% RSLogix 500 project I2P JOB 23 - SOLUTION_BAK116.RSS, saved by version 10.00.00.00 %
PROJECT "MLO2B"    % processor: Bul.1763 MicroLogix 1100 Series B %

PROGRAM FILES
  LAD 2   18 rungs

DATA FILES
  O0 OUTPUT  4 elements
  I1 INPUT  6 elements
  S2 STATUS  66 elements
  B3 BINARY  1 elements
  T4 TIMER  2 elements
  C5 COUNTER  2 elements
  R6 CONTROL  1 elements
  N7 INTEGER  2 elements
  F8 FLOAT  1 elements

LADDER 2
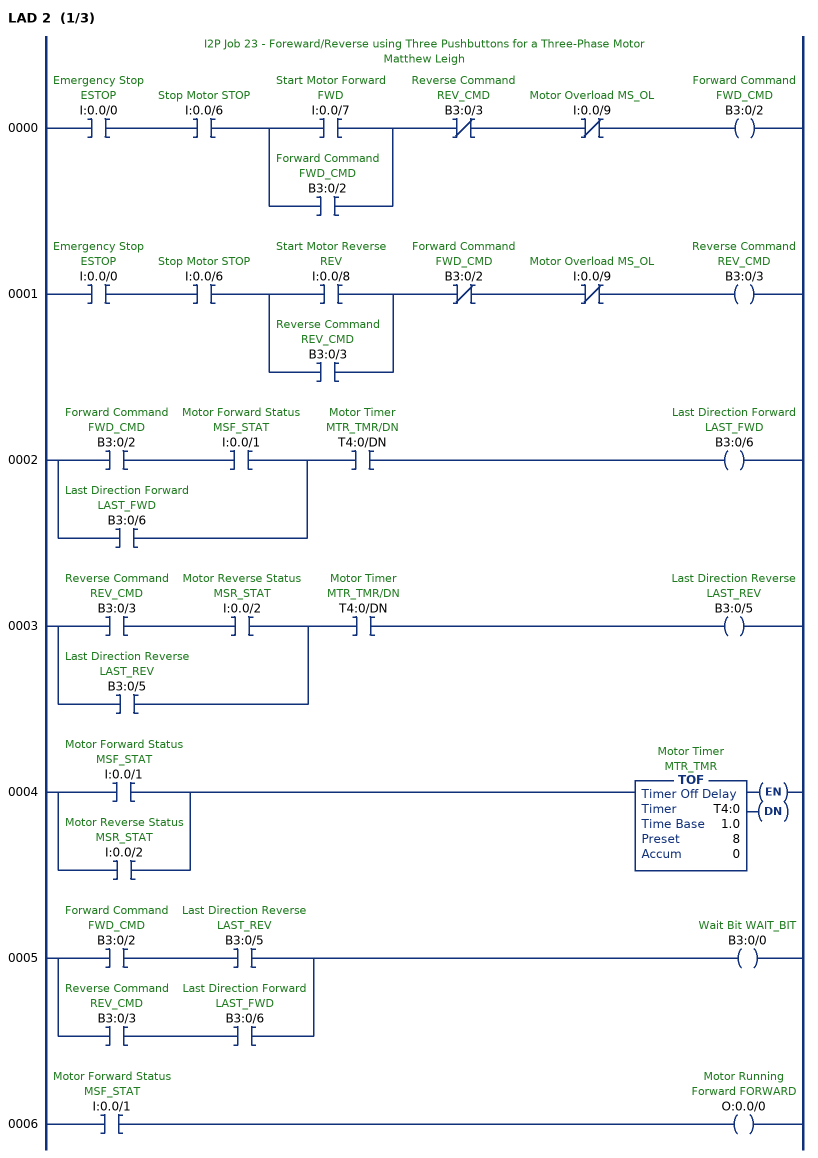
% Rung: 0 %
% I2P Job 23 - Foreward/Reverse using Three Pushbuttons for a Three-Phase Motor
% Matthew Leigh %
SOR XIC I:0.0/0 XIC I:0.0/6 BST XIC I:0.0/7 NXB XIC B3:0/2 BND XIO B3:0/3 XIO I:0.0/9 OTE B3:0/2 EOR
%   I:0.0/0  ESTOP  "Emergency Stop" %
%   I:0.0/6  STOP  "Stop Motor" %
%   I:0.0/7  FWD  "Start Motor Forward" %
%   B3:0/2  FWD_CMD  "Forward Command" %
%   B3:0/3  REV_CMD  "Reverse Command" %
%   I:0.0/9  MS_OL  "Motor Overload" %
% Rung: 1 %
SOR XIC I:0.0/0 XIC I:0.0/6 BST XIC I:0.0/8 NXB XIC B3:0/3 BND XIO B3:0/2 XIO I:0.0/9 OTE B3:0/3 EOR
%   I:0.0/0  ESTOP  "Emergency Stop" %
%   I:0.0/6  STOP  "Stop Motor" %
%   I:0.0/8  REV  "Start Motor Reverse" %
%   B3:0/3  REV_CMD  "Reverse Command" %
%   B3:0/2  FWD_CMD  "Forward Command" %
%   I:0.0/9  MS_OL  "Motor Overload" %
% Rung: 2 %
SOR BST XIC B3:0/2 XIC I:0.0/1 NXB XIC B3:0/6 BND XIC T4:0/DN OTE B3:0/6 EOR
%   B3:0/2  FWD_CMD  "Forward Command" %
%   I:0.0/1  MSF_STAT  "Motor Forward Status" %
%   B3:0/6  LAST_FWD  "Last Direction Forward" %
%   T4:0  MTR_TMR  "Motor Timer" %
% Rung: 3 %
SOR BST XIC B3:0/3 XIC I:0.0/2 NXB XIC B3:0/5 BND XIC T4:0/DN OTE B3:0/5 EOR
%   B3:0/3  REV_CMD  "Reverse Command" %
%   I:0.0/2  MSR_STAT  "Motor Reverse Status" %
%   B3:0/5  LAST_REV  "Last Direction Reverse" %
%   T4:0  MTR_TMR  "Motor Timer" %
% Rung: 4 %
SOR BST XIC I:0.0/1 NXB XIC I:0.0/2 BND TOF T4:0 1.0 8 0 EOR
%   I:0.0/1  MSF_STAT  "Motor Forward Status" %
%   I:0.0/2  MSR_STAT  "Motor Reverse Status" %
%   T4:0  MTR_TMR  "Motor Timer" %
% Rung: 5 %
SOR BST XIC B3:0/2 XIC B3:0/5 NXB XIC B3:0/3 XIC B3:0/6 BND OTE B3:0/0 EOR
%   B3:0/2  FWD_CMD  "Forward Command" %
%   B3:0/5  LAST_REV  "Last Direction Reverse" %
%   B3:0/3  REV_CMD  "Reverse Command" %
%   B3:0/6  LAST_FWD  "Last Direction Forward" %
%   B3:0/0  WAIT_BIT  "Wait Bit" %
% Rung: 6 %
SOR XIC I:0.0/1 OTE O:0.0/0 EOR
%   I:0.0/1  MSF_STAT  "Motor Forward Status" %
%   O:0.0/0  FORWARD  "Motor Running Forward" %

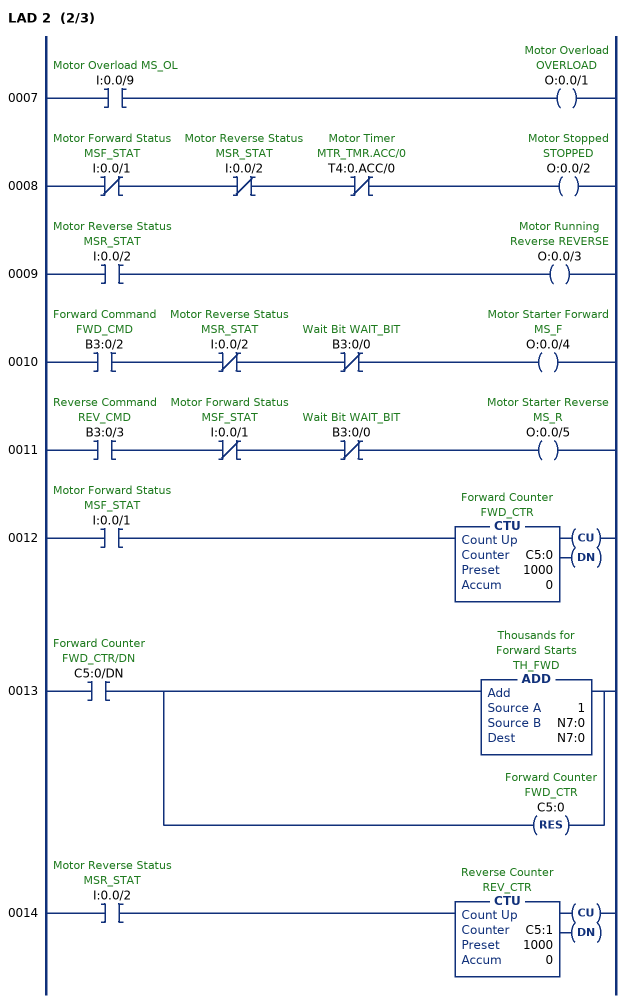
% Rung: 7 %
SOR XIC I:0.0/9 OTE O:0.0/1 EOR
%   I:0.0/9  MS_OL  "Motor Overload" %
%   O:0.0/1  OVERLOAD  "Motor Overload" %
% Rung: 8 %
SOR XIO I:0.0/1 XIO I:0.0/2 XIO T4:0.ACC/0 OTE O:0.0/2 EOR
%   I:0.0/1  MSF_STAT  "Motor Forward Status" %
%   I:0.0/2  MSR_STAT  "Motor Reverse Status" %
%   T4:0  MTR_TMR  "Motor Timer" %
%   O:0.0/2  STOPPED  "Motor Stopped" %
% Rung: 9 %
SOR XIC I:0.0/2 OTE O:0.0/3 EOR
%   I:0.0/2  MSR_STAT  "Motor Reverse Status" %
%   O:0.0/3  REVERSE  "Motor Running Reverse" %
% Rung: 10 %
SOR XIC B3:0/2 XIO I:0.0/2 XIO B3:0/0 OTE O:0.0/4 EOR
%   B3:0/2  FWD_CMD  "Forward Command" %
%   I:0.0/2  MSR_STAT  "Motor Reverse Status" %
%   B3:0/0  WAIT_BIT  "Wait Bit" %
%   O:0.0/4  MS_F  "Motor Starter Forward" %
% Rung: 11 %
SOR XIC B3:0/3 XIO I:0.0/1 XIO B3:0/0 OTE O:0.0/5 EOR
%   B3:0/3  REV_CMD  "Reverse Command" %
%   I:0.0/1  MSF_STAT  "Motor Forward Status" %
%   B3:0/0  WAIT_BIT  "Wait Bit" %
%   O:0.0/5  MS_R  "Motor Starter Reverse" %
% Rung: 12 %
SOR XIC I:0.0/1 CTU C5:0 1000 0 EOR
%   I:0.0/1  MSF_STAT  "Motor Forward Status" %
%   C5:0  FWD_CTR  "Forward Counter" %
% Rung: 13 %
SOR XIC C5:0/DN BST ADD 1 N7:0 N7:0 NXB RES C5:0 BND EOR
%   C5:0  FWD_CTR  "Forward Counter" %
%   N7:0  TH_FWD  "Thousands for Forward Starts" %
% Rung: 14 %
SOR XIC I:0.0/2 CTU C5:1 1000 0 EOR
%   I:0.0/2  MSR_STAT  "Motor Reverse Status" %
%   C5:1  REV_CTR  "Reverse Counter" %

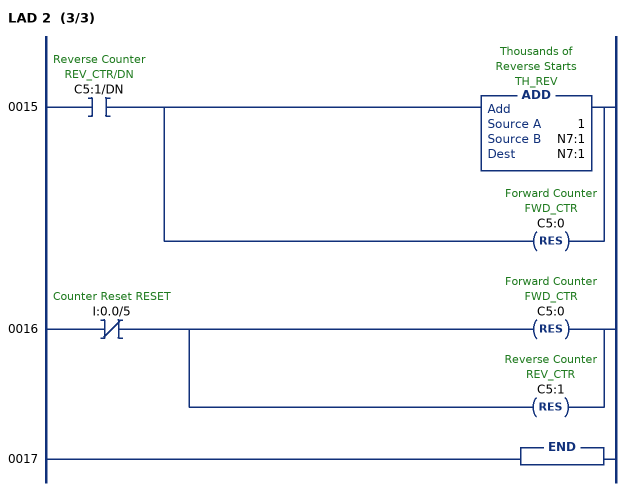
% Rung: 15 %
SOR XIC C5:1/DN BST ADD 1 N7:1 N7:1 NXB RES C5:0 BND EOR
%   C5:1  REV_CTR  "Reverse Counter" %
%   N7:1  TH_REV  "Thousands of Reverse Starts" %
%   C5:0  FWD_CTR  "Forward Counter" %
% Rung: 16 %
SOR XIO I:0.0/5 BST RES C5:0 NXB RES C5:1 BND EOR
%   I:0.0/5  RESET  "Counter Reset" %
%   C5:0  FWD_CTR  "Forward Counter" %
%   C5:1  REV_CTR  "Reverse Counter" %
% Rung: 17 %
SOR END EOR

OTHER DOCUMENTED ADDRESSES
  B3:0/1  ON_BIT  "On position bit"
  B3:0/4  YLW_LT_BIT
  B3:0/7  STOP_BIT  "Estop and Stop"
  FWD_JOG  "Forward Jog"
  I:0.0/3  AUTO_POS  "3 Position Selector Switch A Position"
  I:0.0/4  ON  "3 Position Selector Switch B Position"
  MOTOR  
  T4  
  T4:0/EN  TIMER_ENABLED
  T4:1  FWD_DELAY

DATA TABLE (non-zero values as saved)
DATA B3
% B3:0 % 0X0040
DATA T4
% .PRE .ACC %
% T4:0 % 8 0
% T4:1 % 8 0
DATA C5
% .PRE .ACC %
% C5:0 % 1000 0
% C5:1 % 1000 0
